(* 
:Description: This function is used to merge 5 strings
*)
FUNCTION FUN_MergeStrings3 : STRING
VAR_INPUT
	sStr1	: STRING;			(* Fifth string in merge row *)
	sStr2	: STRING;			(* Fourth string in merge row *)
	sStr3	: STRING;			(* Fourth string in merge row *)

END_VAR

FUN_MergeStrings3 := CONCAT(sStr1,sStr2);
FUN_MergeStrings3 := CONCAT(FUN_MergeStrings3,sStr3);

END_FUNCTION

(* stored: Version 1.1.0.1, ProductVersion 3.1.4024.12
   POU FUN_MergeStrings3: Id {a7dc5695-0618-4375-a202-b8b45cf00675}, SpecialFunc None *)
